FUNCTION Convert_SINT_TO_USINT : BOOL
VAR_INPUT
	in : SINT;
	out : REFERENCE TO USINT;
END_VAR
VAR
	converted : USINT;
END_VAR

converted := SINT_TO_USINT(in);

IF (USINT_TO_SINT(converted) <> in) THEN
	RETURN;
END_IF

out := converted;
Convert_SINT_TO_USINT := TRUE;

END_FUNCTION

(* stored: Version 1.1.0.1, ProductVersion 3.1.4024.12
   POU Convert_SINT_TO_USINT: Id {0cfed76a-70b3-429d-bf14-ea58b536835c}, SpecialFunc None *)
